(* PLC project tapis_conv, TNI-Software ControlBuild 4.00 *)
(* stored: creationDateTime 2018-09-10T16:28:26-01:00 *)

PROGRAM tapis_conv.tapis_conv

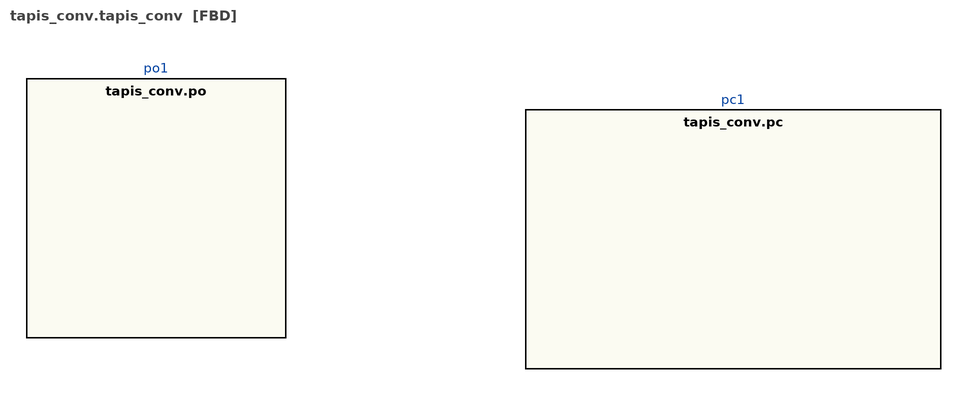
(* FBD diagram, written out as Structured Text *)
po1();
pc1();
END_PROGRAM
